% RSLogix 500 project VILLA_PARK_DRYER_FEB_17_2022.RSS, saved by version 11.00.00.00 %
PROJECT "ML1200"    % processor: MicroLogix 1400; MAIN_PROG %

PROGRAM FILES
  LAD 2 "MAIN_PROG"  7 rungs
  LAD 3   30 rungs
  LAD 4   11 rungs
  LAD 5   24 rungs
  LAD 6   6 rungs
  LAD 7   31 rungs
  LAD 8   5 rungs

DATA FILES
  O0 OUTPUT  10 elements
  I1 INPUT  23 elements
  S2 STATUS  66 elements
  B3 BINARY  3 elements
  T4 TIMER  5 elements
  C5 COUNTER  1 elements
  R6 CONTROL  1 elements
  N7 INTEGER  60 elements
  F8 FLOAT  1 elements
  PD9   2 elements

LADDER 2 "MAIN_PROG"
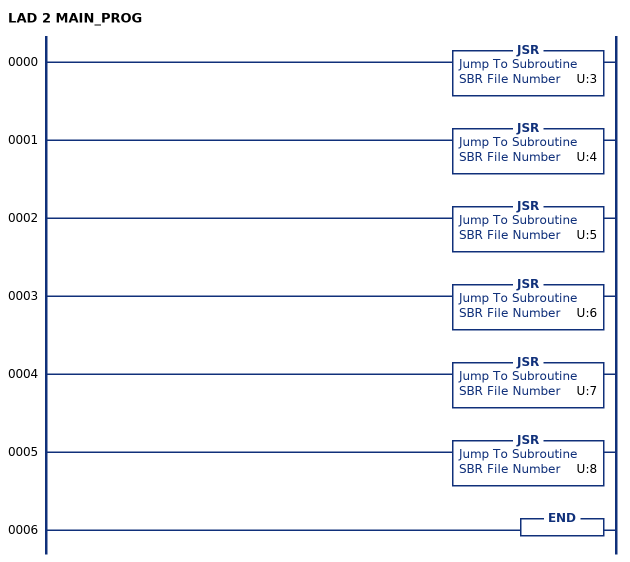
% Rung: 0 %
SOR JSR U:3 EOR
% Rung: 1 %
SOR JSR U:4 EOR
% Rung: 2 %
SOR JSR U:5 EOR
% Rung: 3 %
SOR JSR U:6 EOR
% Rung: 4 %
SOR JSR U:7 EOR
% Rung: 5 %
SOR JSR U:8 EOR
% Rung: 6 %
SOR END EOR

LADDER 3
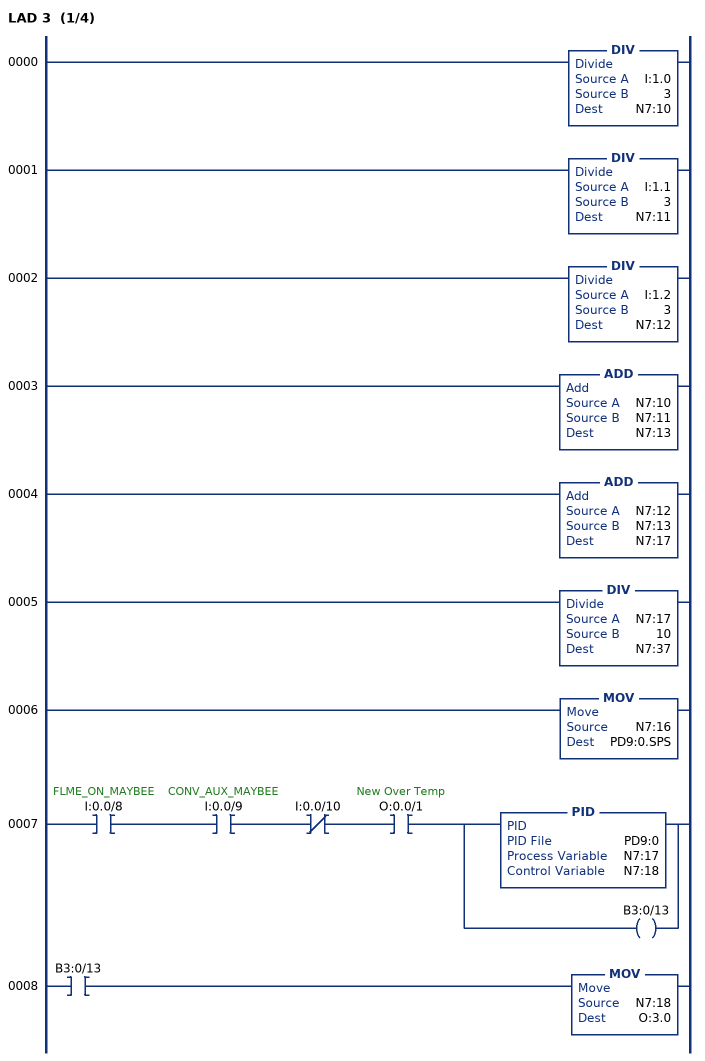
% Rung: 0 %
SOR DIV I:1.0 3 N7:10 EOR
% Rung: 1 %
SOR DIV I:1.1 3 N7:11 EOR
% Rung: 2 %
SOR DIV I:1.2 3 N7:12 EOR
% Rung: 3 %
SOR ADD N7:10 N7:11 N7:13 EOR
% Rung: 4 %
SOR ADD N7:12 N7:13 N7:17 EOR
% Rung: 5 %
SOR DIV N7:17 10 N7:37 EOR
% Rung: 6 %
SOR MOV N7:16 PD9:0.SPS EOR
% Rung: 7 %
SOR XIC I:0.0/8 XIC I:0.0/9 XIO I:0.0/10 XIC O:0.0/1 BST PID PD9:0 N7:17 N7:18 NXB OTE B3:0/13 BND EOR
%   I:0.0/8  FLME_ON_MAYBEE %
%   I:0.0/9  CONV_AUX_MAYBEE %
%   O:0.0/1  "New Over Temp" %
% Rung: 8 %
SOR XIC B3:0/13 MOV N7:18 O:3.0 EOR

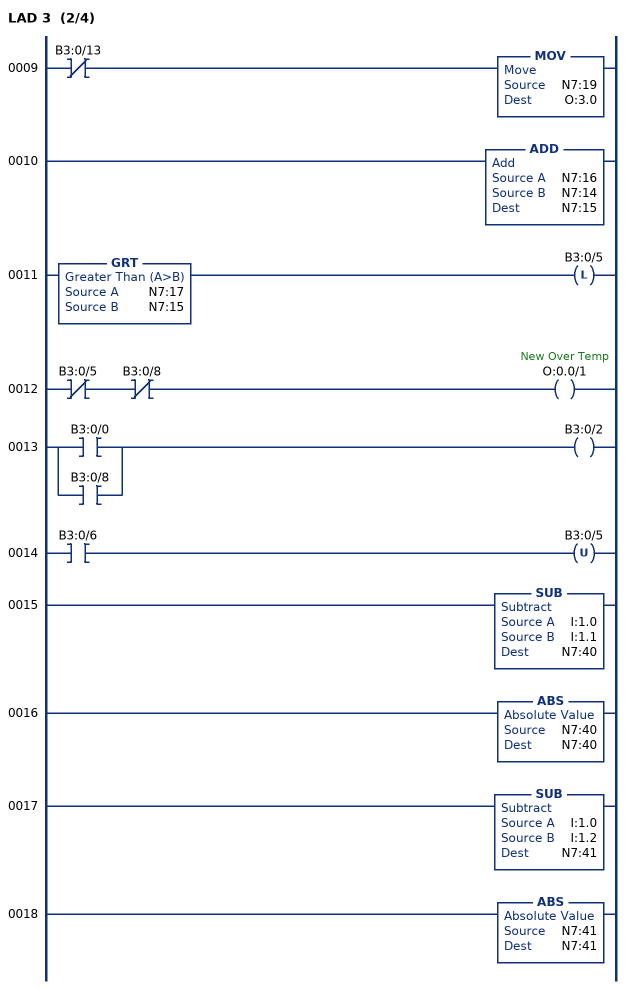
% Rung: 9 %
SOR XIO B3:0/13 MOV N7:19 O:3.0 EOR
% Rung: 10 %
SOR ADD N7:16 N7:14 N7:15 EOR
% Rung: 11 %
SOR GRT N7:17 N7:15 OTL B3:0/5 EOR
% Rung: 12 %
SOR XIO B3:0/5 XIO B3:0/8 OTE O:0.0/1 EOR
%   O:0.0/1  "New Over Temp" %
% Rung: 13 %
SOR BST XIC B3:0/0 NXB XIC B3:0/8 BND OTE B3:0/2 EOR
% Rung: 14 %
SOR XIC B3:0/6 OTU B3:0/5 EOR
% Rung: 15 %
SOR SUB I:1.0 I:1.1 N7:40 EOR
% Rung: 16 %
SOR ABS N7:40 N7:40 EOR
% Rung: 17 %
SOR SUB I:1.0 I:1.2 N7:41 EOR
% Rung: 18 %
SOR ABS N7:41 N7:41 EOR

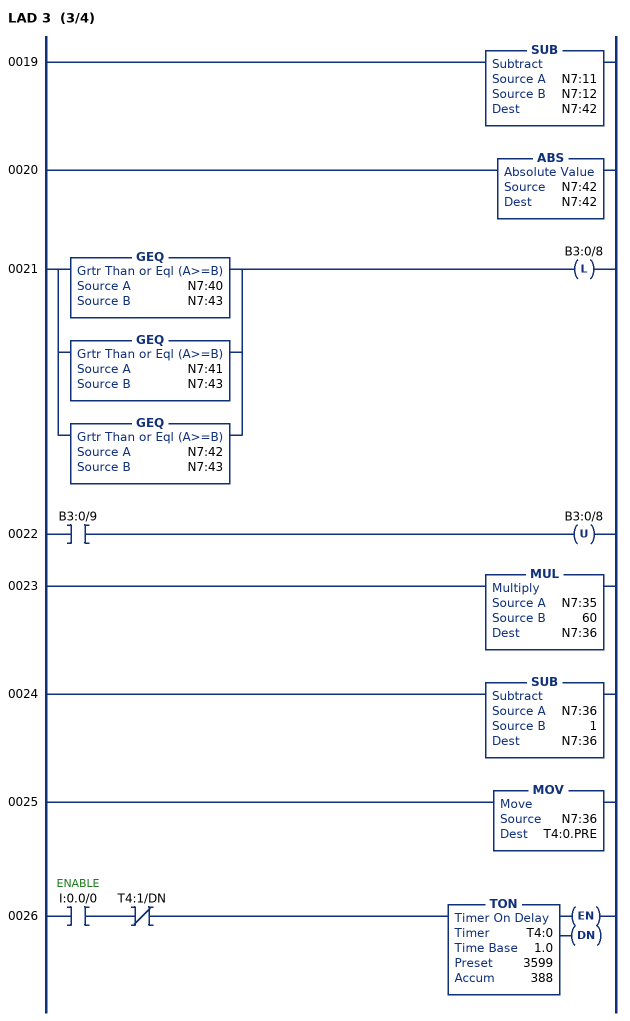
% Rung: 19 %
SOR SUB N7:11 N7:12 N7:42 EOR
% Rung: 20 %
SOR ABS N7:42 N7:42 EOR
% Rung: 21 %
SOR BST GEQ N7:40 N7:43 NXB BST GEQ N7:41 N7:43 NXB GEQ N7:42 N7:43 BND BND OTL B3:0/8 EOR
% Rung: 22 %
SOR XIC B3:0/9 OTU B3:0/8 EOR
% Rung: 23 %
SOR MUL N7:35 60 N7:36 EOR
% Rung: 24 %
SOR SUB N7:36 1 N7:36 EOR
% Rung: 25 %
SOR MOV N7:36 T4:0.PRE EOR
% Rung: 26 %
SOR XIC I:0.0/0 XIO T4:1/DN TON T4:0 1.0 3599 388 EOR
%   I:0.0/0  ENABLE %

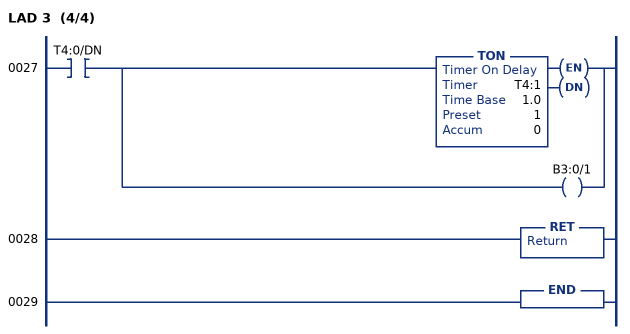
% Rung: 27 %
SOR XIC T4:0/DN BST TON T4:1 1.0 1 0 NXB OTE B3:0/1 BND EOR
% Rung: 28 %
SOR RET EOR
% Rung: 29 %
SOR END EOR

LADDER 4
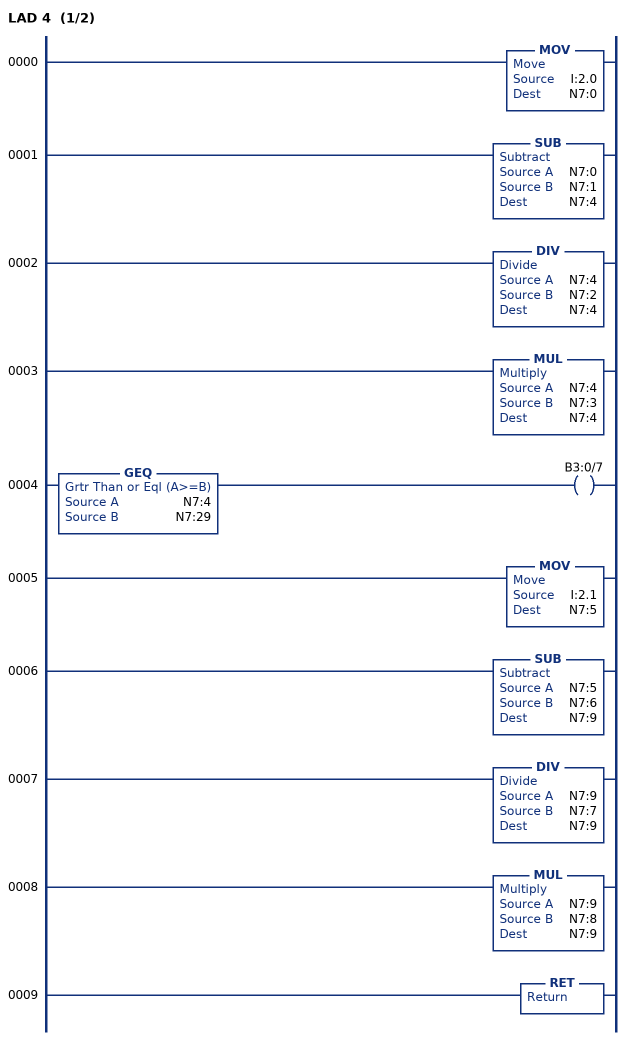
% Rung: 0 %
SOR MOV I:2.0 N7:0 EOR
% Rung: 1 %
SOR SUB N7:0 N7:1 N7:4 EOR
% Rung: 2 %
SOR DIV N7:4 N7:2 N7:4 EOR
% Rung: 3 %
SOR MUL N7:4 N7:3 N7:4 EOR
% Rung: 4 %
SOR GEQ N7:4 N7:29 OTE B3:0/7 EOR
% Rung: 5 %
SOR MOV I:2.1 N7:5 EOR
% Rung: 6 %
SOR SUB N7:5 N7:6 N7:9 EOR
% Rung: 7 %
SOR DIV N7:9 N7:7 N7:9 EOR
% Rung: 8 %
SOR MUL N7:9 N7:8 N7:9 EOR
% Rung: 9 %
SOR RET EOR

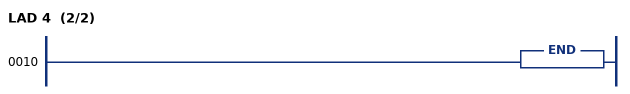
% Rung: 10 %
SOR END EOR

LADDER 5
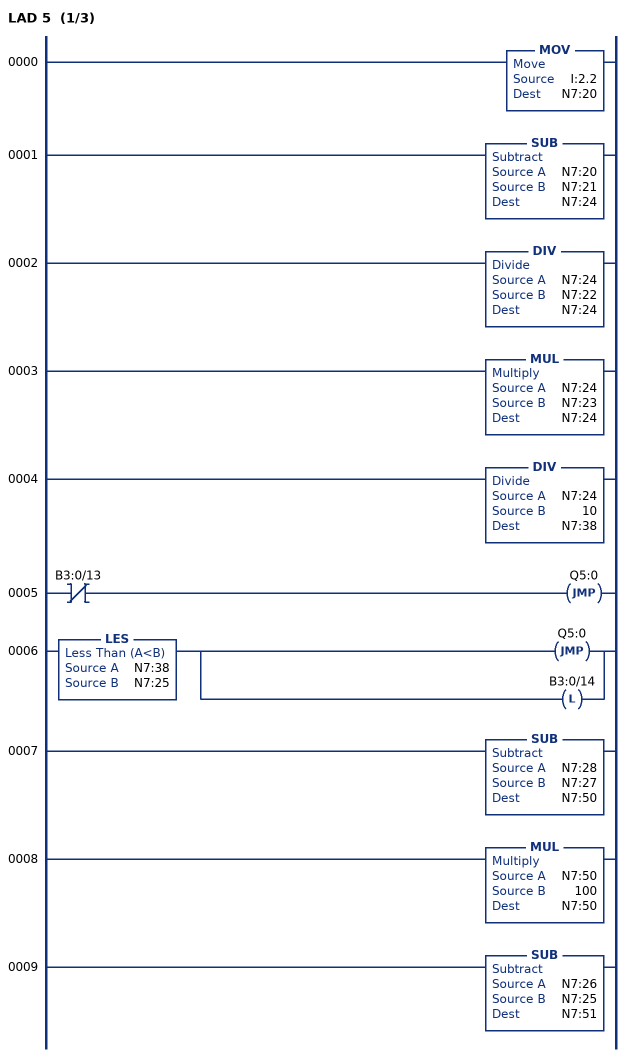
% Rung: 0 %
SOR MOV I:2.2 N7:20 EOR
% Rung: 1 %
SOR SUB N7:20 N7:21 N7:24 EOR
% Rung: 2 %
SOR DIV N7:24 N7:22 N7:24 EOR
% Rung: 3 %
SOR MUL N7:24 N7:23 N7:24 EOR
% Rung: 4 %
SOR DIV N7:24 10 N7:38 EOR
% Rung: 5 %
SOR XIO B3:0/13 JMP Q5:0 EOR
% Rung: 6 %
SOR LES N7:38 N7:25 BST JMP Q5:0 NXB OTL B3:0/14 BND EOR
% Rung: 7 %
SOR SUB N7:28 N7:27 N7:50 EOR
% Rung: 8 %
SOR MUL N7:50 100 N7:50 EOR
% Rung: 9 %
SOR SUB N7:26 N7:25 N7:51 EOR

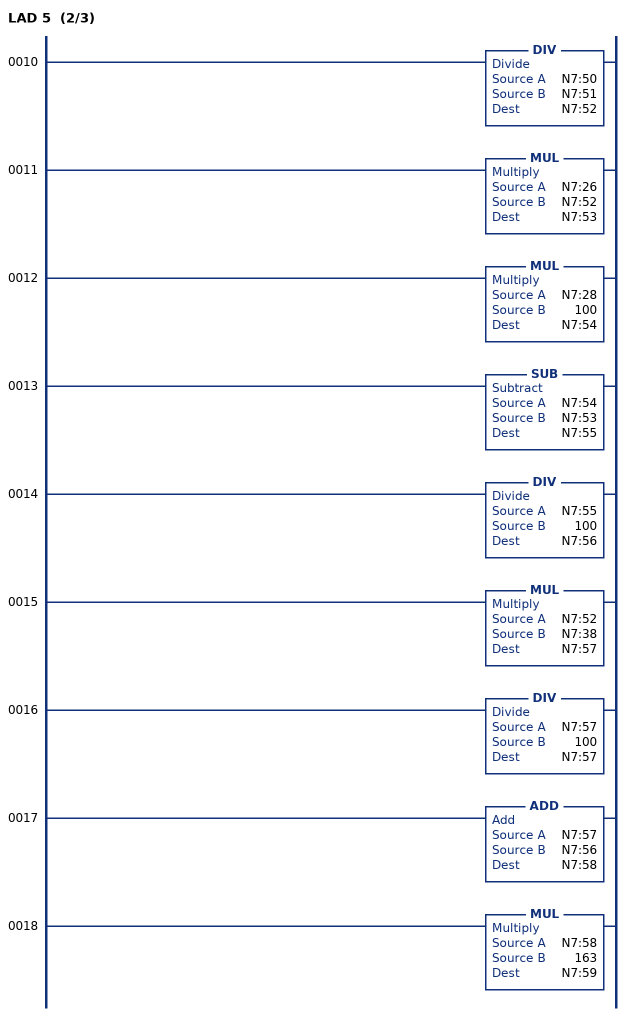
% Rung: 10 %
SOR DIV N7:50 N7:51 N7:52 EOR
% Rung: 11 %
SOR MUL N7:26 N7:52 N7:53 EOR
% Rung: 12 %
SOR MUL N7:28 100 N7:54 EOR
% Rung: 13 %
SOR SUB N7:54 N7:53 N7:55 EOR
% Rung: 14 %
SOR DIV N7:55 100 N7:56 EOR
% Rung: 15 %
SOR MUL N7:52 N7:38 N7:57 EOR
% Rung: 16 %
SOR DIV N7:57 100 N7:57 EOR
% Rung: 17 %
SOR ADD N7:57 N7:56 N7:58 EOR
% Rung: 18 %
SOR MUL N7:58 163 N7:59 EOR

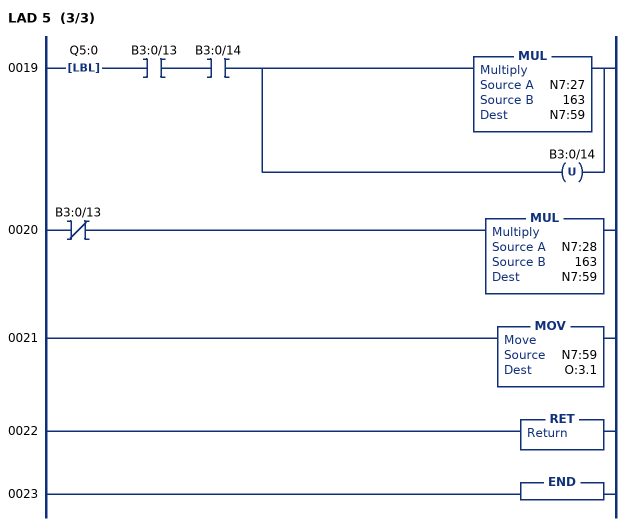
% Rung: 19 %
SOR LBL Q5:0 XIC B3:0/13 XIC B3:0/14 BST MUL N7:27 163 N7:59 NXB OTU B3:0/14 BND EOR
% Rung: 20 %
SOR XIO B3:0/13 MUL N7:28 163 N7:59 EOR
% Rung: 21 %
SOR MOV N7:59 O:3.1 EOR
% Rung: 22 %
SOR RET EOR
% Rung: 23 %
SOR END EOR

LADDER 6
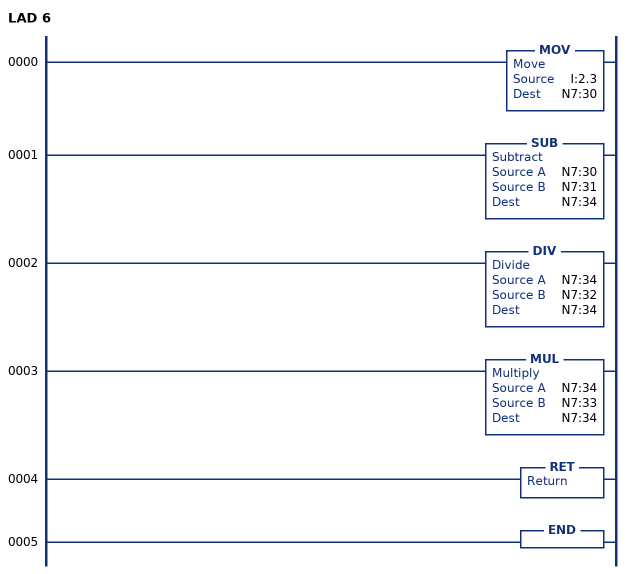
% Rung: 0 %
SOR MOV I:2.3 N7:30 EOR
% Rung: 1 %
SOR SUB N7:30 N7:31 N7:34 EOR
% Rung: 2 %
SOR DIV N7:34 N7:32 N7:34 EOR
% Rung: 3 %
SOR MUL N7:34 N7:33 N7:34 EOR
% Rung: 4 %
SOR RET EOR
% Rung: 5 %
SOR END EOR

LADDER 7
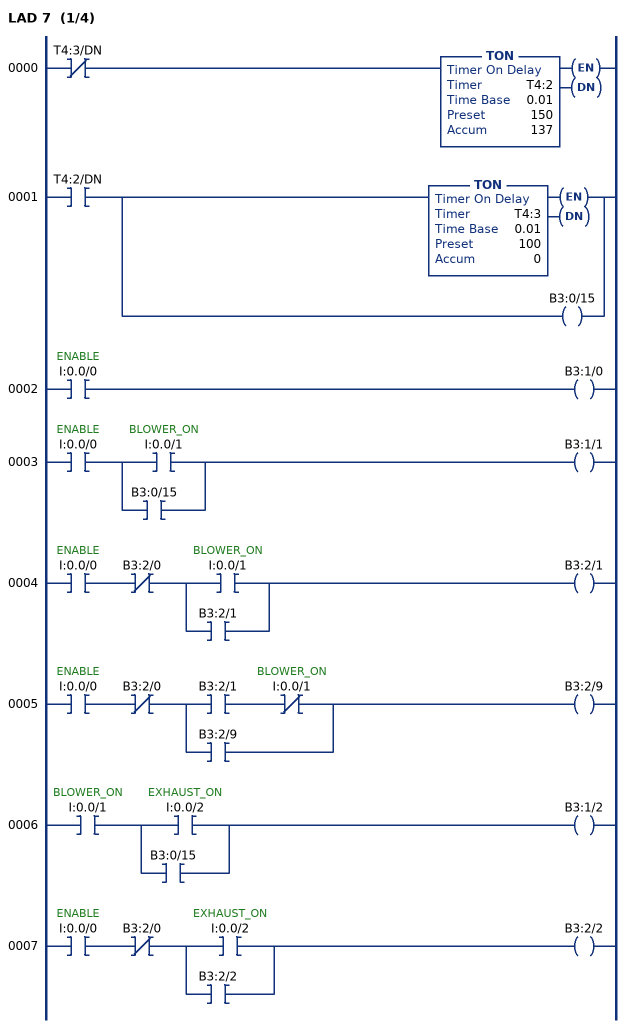
% Rung: 0 %
SOR XIO T4:3/DN TON T4:2 0.01 150 137 EOR
% Rung: 1 %
SOR XIC T4:2/DN BST TON T4:3 0.01 100 0 NXB OTE B3:0/15 BND EOR
% Rung: 2 %
SOR XIC I:0.0/0 OTE B3:1/0 EOR
%   I:0.0/0  ENABLE %
% Rung: 3 %
SOR XIC I:0.0/0 BST XIC I:0.0/1 NXB XIC B3:0/15 BND OTE B3:1/1 EOR
%   I:0.0/0  ENABLE %
%   I:0.0/1  BLOWER_ON %
% Rung: 4 %
SOR XIC I:0.0/0 XIO B3:2/0 BST XIC I:0.0/1 NXB XIC B3:2/1 BND OTE B3:2/1 EOR
%   I:0.0/0  ENABLE %
%   I:0.0/1  BLOWER_ON %
% Rung: 5 %
SOR XIC I:0.0/0 XIO B3:2/0 BST XIC B3:2/1 XIO I:0.0/1 NXB XIC B3:2/9 BND OTE B3:2/9 EOR
%   I:0.0/0  ENABLE %
%   I:0.0/1  BLOWER_ON %
% Rung: 6 %
SOR XIC I:0.0/1 BST XIC I:0.0/2 NXB XIC B3:0/15 BND OTE B3:1/2 EOR
%   I:0.0/1  BLOWER_ON %
%   I:0.0/2  EXHAUST_ON %
% Rung: 7 %
SOR XIC I:0.0/0 XIO B3:2/0 BST XIC I:0.0/2 NXB XIC B3:2/2 BND OTE B3:2/2 EOR
%   I:0.0/0  ENABLE %
%   I:0.0/2  EXHAUST_ON %

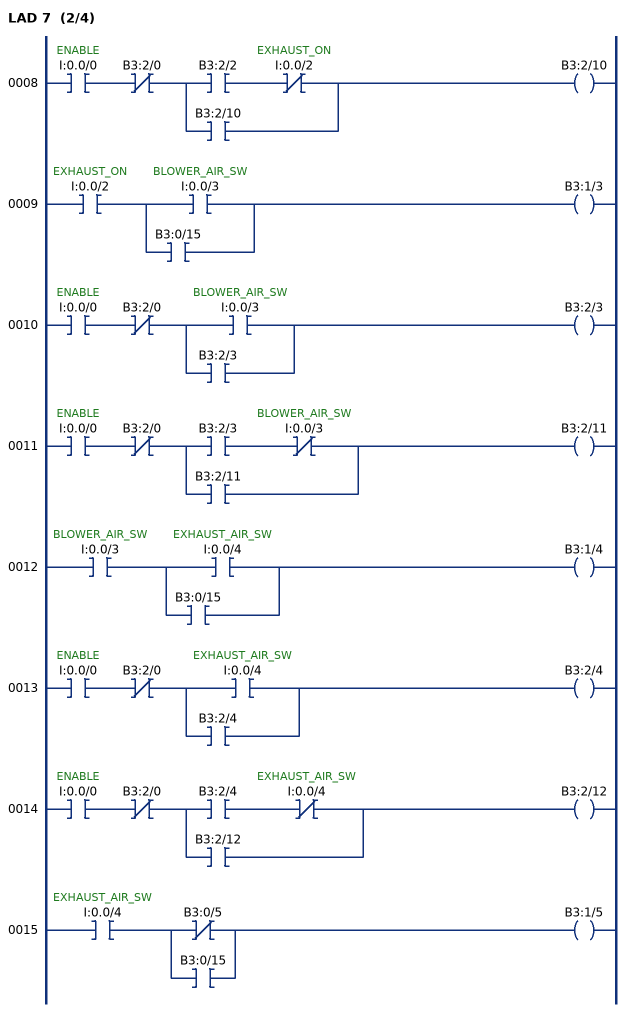
% Rung: 8 %
SOR XIC I:0.0/0 XIO B3:2/0 BST XIC B3:2/2 XIO I:0.0/2 NXB XIC B3:2/10 BND OTE B3:2/10 EOR
%   I:0.0/0  ENABLE %
%   I:0.0/2  EXHAUST_ON %
% Rung: 9 %
SOR XIC I:0.0/2 BST XIC I:0.0/3 NXB XIC B3:0/15 BND OTE B3:1/3 EOR
%   I:0.0/2  EXHAUST_ON %
%   I:0.0/3  BLOWER_AIR_SW %
% Rung: 10 %
SOR XIC I:0.0/0 XIO B3:2/0 BST XIC I:0.0/3 NXB XIC B3:2/3 BND OTE B3:2/3 EOR
%   I:0.0/0  ENABLE %
%   I:0.0/3  BLOWER_AIR_SW %
% Rung: 11 %
SOR XIC I:0.0/0 XIO B3:2/0 BST XIC B3:2/3 XIO I:0.0/3 NXB XIC B3:2/11 BND OTE B3:2/11 EOR
%   I:0.0/0  ENABLE %
%   I:0.0/3  BLOWER_AIR_SW %
% Rung: 12 %
SOR XIC I:0.0/3 BST XIC I:0.0/4 NXB XIC B3:0/15 BND OTE B3:1/4 EOR
%   I:0.0/3  BLOWER_AIR_SW %
%   I:0.0/4  EXHAUST_AIR_SW %
% Rung: 13 %
SOR XIC I:0.0/0 XIO B3:2/0 BST XIC I:0.0/4 NXB XIC B3:2/4 BND OTE B3:2/4 EOR
%   I:0.0/0  ENABLE %
%   I:0.0/4  EXHAUST_AIR_SW %
% Rung: 14 %
SOR XIC I:0.0/0 XIO B3:2/0 BST XIC B3:2/4 XIO I:0.0/4 NXB XIC B3:2/12 BND OTE B3:2/12 EOR
%   I:0.0/0  ENABLE %
%   I:0.0/4  EXHAUST_AIR_SW %
% Rung: 15 %
SOR XIC I:0.0/4 BST XIO B3:0/5 NXB XIC B3:0/15 BND OTE B3:1/5 EOR
%   I:0.0/4  EXHAUST_AIR_SW %

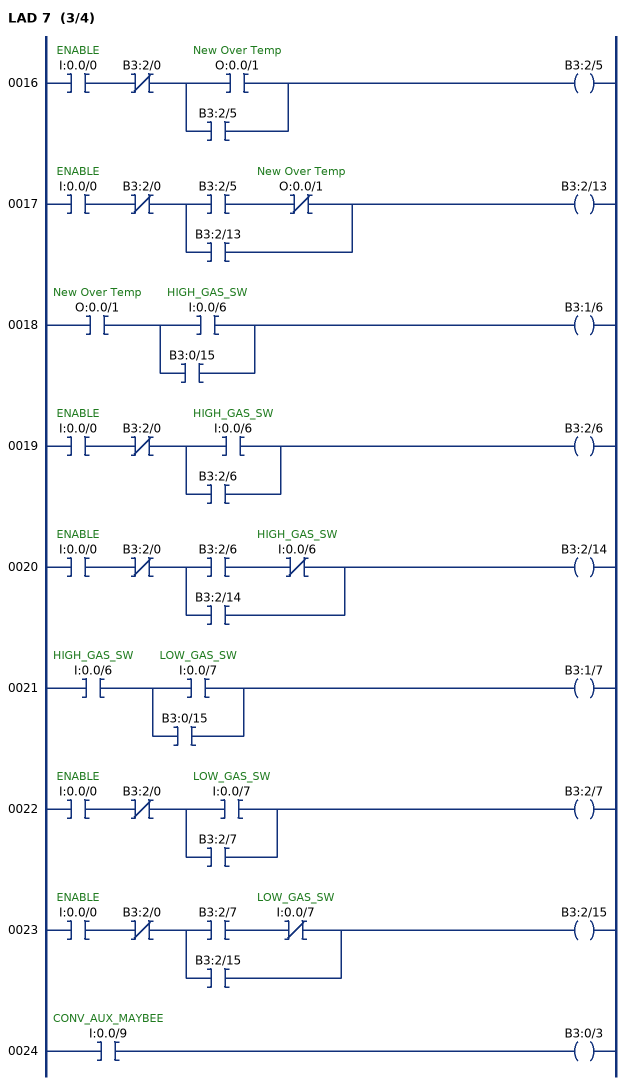
% Rung: 16 %
SOR XIC I:0.0/0 XIO B3:2/0 BST XIC O:0.0/1 NXB XIC B3:2/5 BND OTE B3:2/5 EOR
%   I:0.0/0  ENABLE %
%   O:0.0/1  "New Over Temp" %
% Rung: 17 %
SOR XIC I:0.0/0 XIO B3:2/0 BST XIC B3:2/5 XIO O:0.0/1 NXB XIC B3:2/13 BND OTE B3:2/13 EOR
%   I:0.0/0  ENABLE %
%   O:0.0/1  "New Over Temp" %
% Rung: 18 %
SOR XIC O:0.0/1 BST XIC I:0.0/6 NXB XIC B3:0/15 BND OTE B3:1/6 EOR
%   O:0.0/1  "New Over Temp" %
%   I:0.0/6  HIGH_GAS_SW %
% Rung: 19 %
SOR XIC I:0.0/0 XIO B3:2/0 BST XIC I:0.0/6 NXB XIC B3:2/6 BND OTE B3:2/6 EOR
%   I:0.0/0  ENABLE %
%   I:0.0/6  HIGH_GAS_SW %
% Rung: 20 %
SOR XIC I:0.0/0 XIO B3:2/0 BST XIC B3:2/6 XIO I:0.0/6 NXB XIC B3:2/14 BND OTE B3:2/14 EOR
%   I:0.0/0  ENABLE %
%   I:0.0/6  HIGH_GAS_SW %
% Rung: 21 %
SOR XIC I:0.0/6 BST XIC I:0.0/7 NXB XIC B3:0/15 BND OTE B3:1/7 EOR
%   I:0.0/6  HIGH_GAS_SW %
%   I:0.0/7  LOW_GAS_SW %
% Rung: 22 %
SOR XIC I:0.0/0 XIO B3:2/0 BST XIC I:0.0/7 NXB XIC B3:2/7 BND OTE B3:2/7 EOR
%   I:0.0/0  ENABLE %
%   I:0.0/7  LOW_GAS_SW %
% Rung: 23 %
SOR XIC I:0.0/0 XIO B3:2/0 BST XIC B3:2/7 XIO I:0.0/7 NXB XIC B3:2/15 BND OTE B3:2/15 EOR
%   I:0.0/0  ENABLE %
%   I:0.0/7  LOW_GAS_SW %
% Rung: 24 %
SOR XIC I:0.0/9 OTE B3:0/3 EOR
%   I:0.0/9  CONV_AUX_MAYBEE %

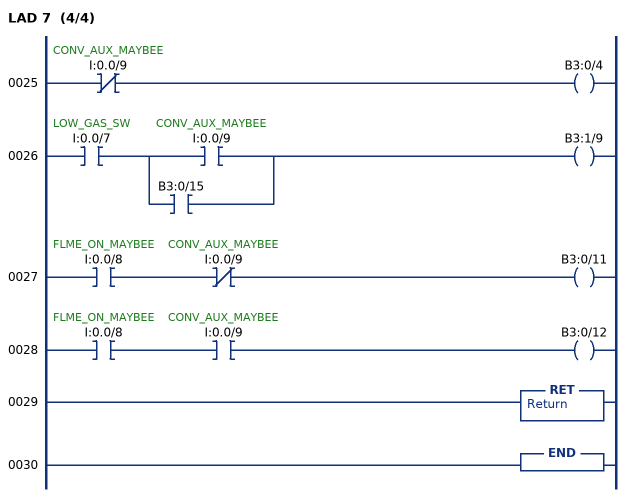
% Rung: 25 %
SOR XIO I:0.0/9 OTE B3:0/4 EOR
%   I:0.0/9  CONV_AUX_MAYBEE %
% Rung: 26 %
SOR XIC I:0.0/7 BST XIC I:0.0/9 NXB XIC B3:0/15 BND OTE B3:1/9 EOR
%   I:0.0/7  LOW_GAS_SW %
%   I:0.0/9  CONV_AUX_MAYBEE %
% Rung: 27 %
SOR XIC I:0.0/8 XIO I:0.0/9 OTE B3:0/11 EOR
%   I:0.0/8  FLME_ON_MAYBEE %
%   I:0.0/9  CONV_AUX_MAYBEE %
% Rung: 28 %
SOR XIC I:0.0/8 XIC I:0.0/9 OTE B3:0/12 EOR
%   I:0.0/8  FLME_ON_MAYBEE %
%   I:0.0/9  CONV_AUX_MAYBEE %
% Rung: 29 %
SOR RET EOR
% Rung: 30 %
SOR END EOR

LADDER 8
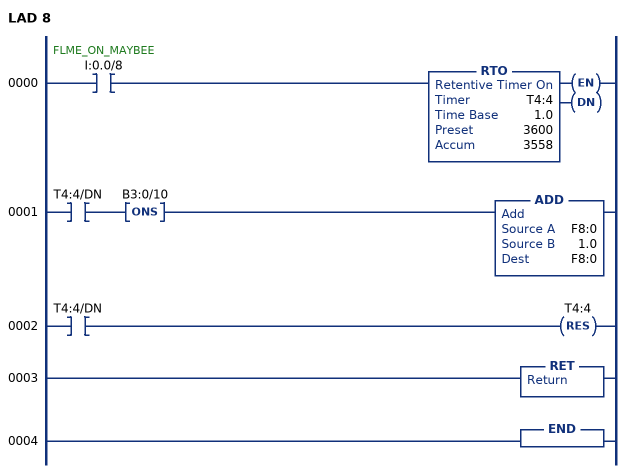
% Rung: 0 %
SOR XIC I:0.0/8 RTO T4:4 1.0 3600 3558 EOR
%   I:0.0/8  FLME_ON_MAYBEE %
% Rung: 1 %
SOR XIC T4:4/DN ONS B3:0/10 ADD F8:0 1.0 F8:0 EOR
% Rung: 2 %
SOR XIC T4:4/DN RES T4:4 EOR
% Rung: 3 %
SOR RET EOR
% Rung: 4 %
SOR END EOR

OTHER DOCUMENTED ADDRESSES
  I:0.0/5  UNKOWN

DATA TABLE (non-zero values as saved)
DATA B3
% B3:0 % 0X1028 0X029F 0XE0FE
DATA T4
% .PRE .ACC %
% T4:0 % 3599 388
% T4:1 % 1 0
% T4:2 % 150 137
% T4:3 % 100 0
% T4:4 % 3600 3558
DATA N7
% N7:0 % 3623 3079 65 1 8 3134 3130 7 1 1
% N7:10 % 428 430 418 858 50 1300 1250 1276 6148 8000
% N7:20 % 11996 3110 115 10 770 25 100 80 100 12
% N7:30 % 3 3110 8 1 -388 60 3599 128 77 0
% N7:40 % 6 31 12 120 0 0 0 0 0 0
% N7:50 % 2000 75 27 2700 10000 7300 73 21 94 16300
DATA F8
% F8:0 % 22612
